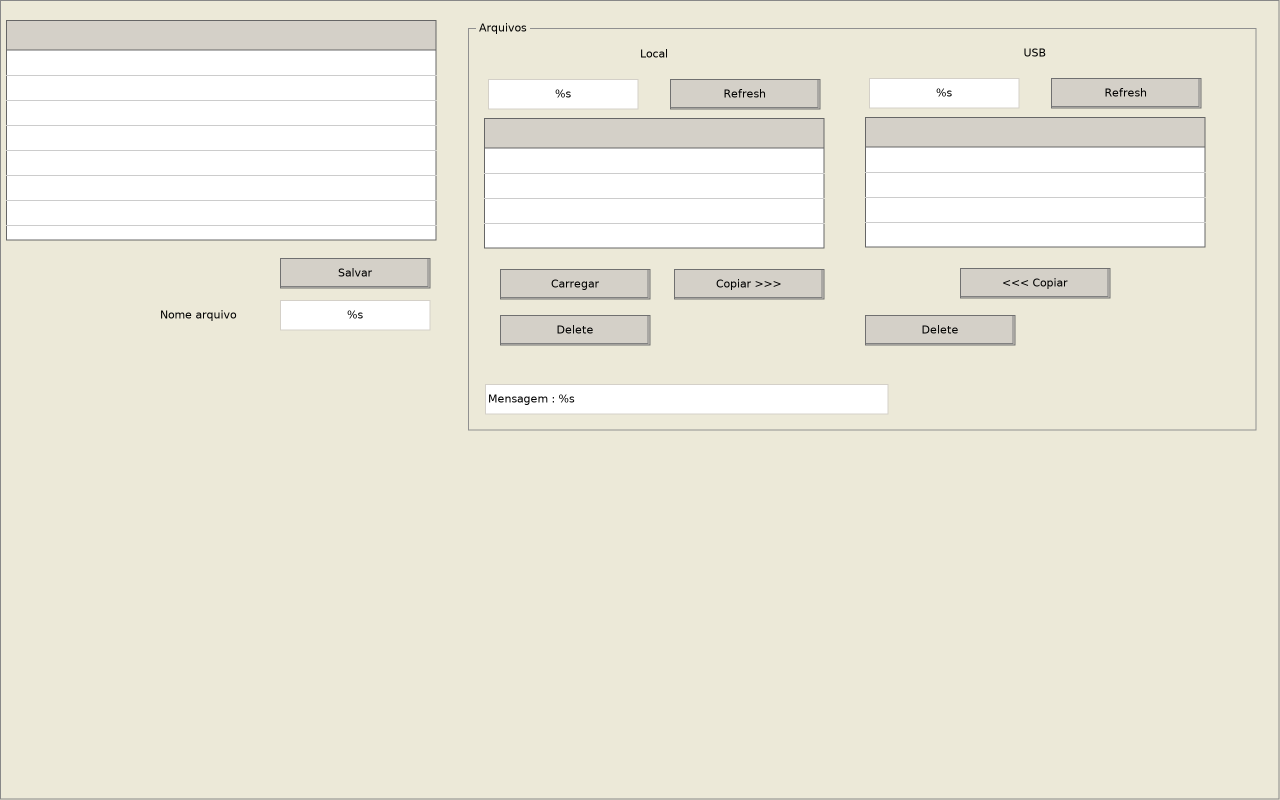
VISUALIZATION Visualization  // 1280x800
    Table (6,20 430x220), data array: MAIN.aStructs
        p3854506369: MAIN.aStructs[INDEX].r1
        p1892666644: MAIN.aStructs[INDEX].i1
        p338671338: MAIN.aStructs[INDEX].s1
        p2170511999: MAIN.aStructs[INDEX].s2
        p3723444502: MAIN.aStructs[INDEX].r2
        p1218418051: MAIN.aStructs[INDEX].i2
    Button (280,258 150x30), "Salvar"
        tap prgFileHnd.bWrite
    Label (144,300 109x30), "Nome arquivo"
    Textfield (280,300 150x30), "%s", text variable: prgFileHnd.sFileName
        OnMouseClick: write the text variable via Default
    GroupBox (468,20 788x410), "Arquivos"
        Table (16,98 340x130), data array: prgFileManipulation.filesInfo
            p3854506369: prgFileManipulation.filesInfo[INDEX].fileName
            p1892666644: prgFileManipulation.filesInfo[INDEX].dataCriacao
            p2232123230: Nome
            p511219082: Criação
            p1137915858: prgFileManipulation.selectedRowLocal
        Textfield (20,59 150x30), "%s", text variable: prgFileManipulation.path
            OnMouseClick: write the text variable via Default
        Button (202,59 150x30), "Refresh"
            tap prgFileManipulation.bFindFiles
        Label (111,19 150x30), "Local"
        Table (397,97 340x130), data array: prgFileManipulation.filesInfoUSB
            p3854506369: prgFileManipulation.filesInfoUSB[INDEX].fileName
            p1892666644: prgFileManipulation.filesInfoUSB[INDEX].dataCriacao
            p2232123230: Nome
            p511219082: Criação
            p1137915858: prgFileManipulation.selectedRowUSB
        Button (206,249 150x30), "Copiar >>>"
            tap prgFileManipulation.copyLocalTOUSB
        Button (492,248 150x30), "<<< Copiar"
            tap prgFileManipulation.copyUSBToLocal
        Textfield (17,364 403x30), "Mensagem : %s", text variable: prgFileManipulation.sCopyMsg
        Button (32,249 150x30), "Carregar"
            tap prgFileHnd.bRead
        Button (32,295 150x30), "Delete"
            tap prgFileManipulation.deleteLocalFile
        Button (397,295 150x30), "Delete"
            tap prgFileManipulation.deleteUSBFile
    Textfield (869,78 150x30), "%s", text variable: prgFileManipulation.pathUSB
        OnMouseClick: write the text variable via Default
    Button (1051,78 150x30), "Refresh"
        tap prgFileManipulation.bFindFilesUSB
    Label (960,38 150x30), "USB"
END_VISUALIZATION

(* stored: Version 1.1.0.1, ProductVersion 3.1.4024.12
   Visu Visualization: Id {254750a9-d74e-445f-b61a-927d675cf0be} *)
